{attribute addProperty BoxType "EL3164-0000-0020"}
{attribute addProperty Id "AI_Standard_Channel_1AT %I*AI_Standard_Channel_BDD14BAD10AI_Compact_Channel_2AT %I*AI_Compact_Channel_80E77D6A2AI_Standard_Channel_3AT %I*AI_Standard_Channel_BDD14BAD10AI_Compact_Channel_4AT %I*AI_Compact_Channel_80E77D6A2WcStateAT %I*WcState_9091E0EB2InfoDataAT %I*InfoData_32EB74EA10"}
{attribute addProperty CRC "1202982053"}
{attribute addProperty SizeInBites "288"}
{attribute addProperty SizeInBytes "36"}
TYPE EL3164_47B40CA5 :
STRUCT
	{attribute addProperty Name "AI_Standard_Channel_1"}
	AI_Standard_Channel_1 : AI_Standard_Channel_BDD14BAD;
	{attribute addProperty Name "AI_Compact_Channel_2"}
	AI_Compact_Channel_2 : AI_Compact_Channel_80E77D6A;
	{attribute addProperty Name "AI_Standard_Channel_3"}
	AI_Standard_Channel_3 : AI_Standard_Channel_BDD14BAD;
	{attribute addProperty Name "AI_Compact_Channel_4"}
	AI_Compact_Channel_4 : AI_Compact_Channel_80E77D6A;
	{attribute addProperty Name "WcState"}
	WcState : WcState_9091E0EB;
	{attribute addProperty Name "InfoData"}
	InfoData : InfoData_32EB74EA;
END_STRUCT
END_TYPE

(* stored: Version 1.2.0.0, ProductVersion 3.1.4024.9
   DUT EL3164_47B40CA5: Id {7af2beb7-2082-41f3-8986-7d304aec6f74} *)
